Staubli VAL3: OnF7.pgx

program OnF7()
begin
  //
  libSave()
  popUpMsg("保存完毕!")
end
